VISUALIZATION VISU_State_gray_orange  // 12x17
VAR_IN_OUT
	state : BOOL;
END_VAR
    Ellipse (0,5 10x10), colour toggle: state
END_VISUALIZATION

(* stored: Version 1.1.0.1, ProductVersion 3.1.0.36
   Visu VISU_State_gray_orange: Id {332063bc-efe6-4ec6-aad0-0769f9248e16} *)
